FUNCTION makeArray0 : ARRAY[0..3] OF DINT
VAR_INPUT
	elem0: DINT;
	elem1: DINT;
	elem2: DINT;
	elem3: DINT;
END_VAR
VAR
	rslt: ARRAY[0..3] OF DINT;
END_VAR

rslt[0] := elem0;
rslt[1] := elem1;
rslt[2] := elem2;
rslt[3] := elem3;
makeArray0 := rslt;

END_FUNCTION

(* stored: Version 1.1.0.1, ProductVersion 3.1.4022.18
   POU makeArray0: Id {8a74912b-ad34-4196-a72f-8800a8287164}, SpecialFunc None *)
